(* IEC 61131-3 sources: axopen.integrations.hwc/app/SystemConstants, 2 files *)

(* ---- plc_line_HwIdentifiers.st ---- *)
CONFIGURATION HardwareIDs
    VAR_GLOBAL CONSTANT
        BNIPNT507005Z040_HwID : UINT := UINT#394;
        BNIPNT507005Z040_BIS_M_4XX_045_1_BIS_M_4XX_045_HwID : UINT := UINT#397;
        BNIPNT507005Z040_BNIPNT507005Z040_HwID : UINT := UINT#396;
        BNIPNT507005Z040_BNIPNT507005Z040_BNI_PNT_507_005_Z040_HwID : UINT := UINT#401;
        BNIPNT507005Z040_BNIPNT507005Z040_profinet_HwID : UINT := UINT#391;
        BNIPNT507005Z040_BNIPNT507005Z040_profinet_port_1___M12_HwID : UINT := UINT#392;
        BNIPNT507005Z040_BNIPNT507005Z040_profinet_port_2___M12_HwID : UINT := UINT#393;
        BNIPNT507005Z040_Rack_HwID : UINT := UINT#395;
        BNIPNT507005Z040_Standard_I_O_2_Standard_I_O_HwID : UINT := UINT#400;
        BNIPNT507005Z040_Standard_I_O_3_Standard_I_O_HwID : UINT := UINT#399;
        BNIPNT507005Z040_Standard_I_O_4_Standard_I_O_HwID : UINT := UINT#398;
        KRC4_HwID : UINT := UINT#467;
        KRC4_512_digital_in_and_outputs_1_512_digital_in__and_outputs_HwID : UINT := UINT#470;
        KRC4_KRC4_HwID : UINT := UINT#469;
        KRC4_KRC4_KRC4_ProfiNet_5_0_HwID : UINT := UINT#471;
        KRC4_KRC4_profinet_HwID : UINT := UINT#465;
        KRC4_KRC4_profinet_Port1_HwID : UINT := UINT#466;
        KRC4_Rack_HwID : UINT := UINT#468;
        OmniCore_HwID : UINT := UINT#337;
        OmniCore_DI_64_bytes_DI_64_bytes_HwID : UINT := UINT#341;
        OmniCore_DO_64_bytes_DO_64_bytes_HwID : UINT := UINT#340;
        OmniCore_OmniCore_HwID : UINT := UINT#339;
        OmniCore_OmniCore_OmniCore_Standard_PROFINET_Device_HwID : UINT := UINT#342;
        OmniCore_OmniCore_profinet_HwID : UINT := UINT#335;
        OmniCore_OmniCore_profinet_Network_Port_1_HwID : UINT := UINT#336;
        OmniCore_Rack_HwID : UINT := UINT#338;
        PROFINET_IO_System_HwID : UINT := UINT#256;
        RobotBasicIO_HwID : UINT := UINT#345;
        RobotBasicIO_DI_64_bytes_DI_64_bytes_HwID : UINT := UINT#349;
        RobotBasicIO_DO_64_bytes_DO_64_bytes_HwID : UINT := UINT#348;
        RobotBasicIO_Rack_HwID : UINT := UINT#346;
        RobotBasicIO_RobotBasicIO_HwID : UINT := UINT#347;
        RobotBasicIO_RobotBasicIO_Robot_Basic_Device_HwID : UINT := UINT#350;
        RobotBasicIO_RobotBasicIO_profinet_HwID : UINT := UINT#343;
        RobotBasicIO_RobotBasicIO_profinet_Network_Port_HwID : UINT := UINT#344;
        SFK_HwID : UINT := UINT#305;
        SFK_F_Modul_not_used_1_ID_FMod_NotUsed_HwID : UINT := UINT#311;
        SFK_Input_24_Words_ID_InMod_24Words_HwID : UINT := UINT#309;
        SFK_Output_21_Words_ID_OutMod_21Words_HwID : UINT := UINT#308;
        SFK_ParamCh_IDN_1_ID_PaCh_5Words_HwID : UINT := UINT#310;
        SFK_Rack_HwID : UINT := UINT#306;
        SFK_SFK_HwID : UINT := UINT#307;
        SFK_SFK_DAP_1_HwID : UINT := UINT#312;
        SFK_SFK_profinet_HwID : UINT := UINT#302;
        SFK_SFK_profinet_Port_1___RJ45_HwID : UINT := UINT#303;
        SFK_SFK_profinet_Port_2___RJ45_HwID : UINT := UINT#304;
        ST3_indradrive_HwID : UINT := UINT#293;
        ST3_indradrive_F_Modul_not_used_1_ID_FMod_NotUsed_HwID : UINT := UINT#299;
        ST3_indradrive_Input_9_Words_1_ID_InMod_9Words_HwID : UINT := UINT#297;
        ST3_indradrive_Output_13_Words_1_ID_OutMod_13Words_HwID : UINT := UINT#296;
        ST3_indradrive_ParamCh_IDN_1_ID_PaCh_5Words_HwID : UINT := UINT#298;
        ST3_indradrive_Rack_HwID : UINT := UINT#294;
        ST3_indradrive_ST3_indradrive_HwID : UINT := UINT#295;
        ST3_indradrive_ST3_indradrive_DAP_1_HwID : UINT := UINT#300;
        ST3_indradrive_ST3_indradrive_profinet_HwID : UINT := UINT#290;
        ST3_indradrive_ST3_indradrive_profinet_Port_1___RJ45_HwID : UINT := UINT#291;
        ST3_indradrive_ST3_indradrive_profinet_Port_2___RJ45_HwID : UINT := UINT#292;
        TZ535_PN_HwID : UINT := UINT#316;
        TZ535_PN_In_Out_64_byte_1_In_Out__64_byte_HwID : UINT := UINT#319;
        TZ535_PN_Rack_HwID : UINT := UINT#317;
        TZ535_PN_TZ535_PN_HwID : UINT := UINT#318;
        TZ535_PN_TZ535_PN_2D_TZ535_PNPROFINET_IO_HwID : UINT := UINT#320;
        TZ535_PN_TZ535_PN_profinet_HwID : UINT := UINT#313;
        TZ535_PN_TZ535_PN_profinet_Port_1_HwID : UINT := UINT#314;
        TZ535_PN_TZ535_PN_profinet_Port_2_HwID : UINT := UINT#315;
        URIODev1_HwID : UINT := UINT#276;
        URIODev1_1_HwID : UINT := UINT#259;
        URIODev1_1_10_O2T_General_Purpose_Registers_2_1_10_O2T_General_Purpose_Registers_2_HwID : UINT := UINT#262;
        URIODev1_1_1_T2O_State_1_1_T2O_State_HwID : UINT := UINT#271;
        URIODev1_1_2_T2O_IO_1_2_T2O_IO_HwID : UINT := UINT#270;
        URIODev1_1_3_T2O_Joints_1_3_T2O_Joints_HwID : UINT := UINT#269;
        URIODev1_1_4_T2O_TCP_1_4_T2O_TCP_HwID : UINT := UINT#268;
        URIODev1_1_5_T2O_General_Purpose_Bit_Registers_1_5_T2O_General_Purpose_Bit_Registers_HwID : UINT := UINT#267;
        URIODev1_1_6_T2O_General_Purpose_Int_Registers_1_6_T2O_General_Purpose_Int_Registers_HwID : UINT := UINT#266;
        URIODev1_1_7_T2O_General_Purpose_Float_Registers_1_7_T2O_General_Purpose_Float_Registers_HwID : UINT := UINT#265;
        URIODev1_1_8_O2T_Robot_IO_1_8_O2T_Robot_IO_HwID : UINT := UINT#264;
        URIODev1_1_9_O2T_General_Purpose_Registers_1_1_9_O2T_General_Purpose_Registers_1_HwID : UINT := UINT#263;
        URIODev1_1_PROFIsafe_1_Module_Access_Point_HwID : UINT := UINT#272;
        URIODev1_1_Rack_HwID : UINT := UINT#260;
        URIODev1_1_URIODev1_1_HwID : UINT := UINT#261;
        URIODev1_1_URIODev1_1_V1_0_HwID : UINT := UINT#273;
        URIODev1_1_URIODev1_1_profinet_HwID : UINT := UINT#257;
        URIODev1_1_URIODev1_1_profinet_RJ45_10_100_MBit_s_HwID : UINT := UINT#258;
        URIODev1_10_O2T_General_Purpose_Registers_2_1_10_O2T_General_Purpose_Registers_2_HwID : UINT := UINT#279;
        URIODev1_1_T2O_State_1_1_T2O_State_HwID : UINT := UINT#288;
        URIODev1_2_T2O_IO_1_2_T2O_IO_HwID : UINT := UINT#287;
        URIODev1_3_T2O_Joints_1_3_T2O_Joints_HwID : UINT := UINT#286;
        URIODev1_4_T2O_TCP_1_4_T2O_TCP_HwID : UINT := UINT#285;
        URIODev1_5_T2O_General_Purpose_Bit_Registers_1_5_T2O_General_Purpose_Bit_Registers_HwID : UINT := UINT#284;
        URIODev1_6_T2O_General_Purpose_Int_Registers_1_6_T2O_General_Purpose_Int_Registers_HwID : UINT := UINT#283;
        URIODev1_7_T2O_General_Purpose_Float_Registers_1_7_T2O_General_Purpose_Float_Registers_HwID : UINT := UINT#282;
        URIODev1_8_O2T_Robot_IO_1_8_O2T_Robot_IO_HwID : UINT := UINT#281;
        URIODev1_9_O2T_General_Purpose_Registers_1_1_9_O2T_General_Purpose_Registers_1_HwID : UINT := UINT#280;
        URIODev1_Rack_HwID : UINT := UINT#277;
        URIODev1_URIODev1_HwID : UINT := UINT#278;
        URIODev1_URIODev1_V1_0_HwID : UINT := UINT#289;
        URIODev1_URIODev1_profinet_HwID : UINT := UINT#274;
        URIODev1_URIODev1_profinet_RJ45_10_100_MBit_s_HwID : UINT := UINT#275;
        aventics_HwID : UINT := UINT#405;
        aventics_Rack_HwID : UINT := UINT#406;
        aventics_Valve_driver_2_valves_1_Valve_driver_2_valves_2_HwID : UINT := UINT#408;
        aventics_Valve_driver_3_valves_1_Valve_driver_3_valves_3_HwID : UINT := UINT#411;
        aventics_Valve_driver_4_valves_1_Valve_driver_4_valves_4_HwID : UINT := UINT#412;
        aventics_Valve_driver_4_valves_2_Valve_driver_4_valves_4_HwID : UINT := UINT#410;
        aventics_Valve_driver_4_valves_3_Valve_driver_4_valves_4_HwID : UINT := UINT#409;
        aventics_aventics_HwID : UINT := UINT#407;
        aventics_aventics_AES_Modul_HwID : UINT := UINT#413;
        aventics_aventics_profinet_HwID : UINT := UINT#402;
        aventics_aventics_profinet_Port_1_HwID : UINT := UINT#403;
        aventics_aventics_profinet_Port_2_HwID : UINT := UINT#404;
        cmmtas_HwID : UINT := UINT#456;
        cmmtas_Rack_HwID : UINT := UINT#457;
        cmmtas_SiemensTelegram111_PZD_12_12_HwID : UINT := UINT#462;
        cmmtas_SiemensTelegram750_PZD_4_1_HwID : UINT := UINT#463;
        cmmtas_cmmtas_HwID : UINT := UINT#458;
        cmmtas_cmmtas_CMMT_AS_____MP_HwID : UINT := UINT#464;
        cmmtas_cmmtas_DoServo_HwID : UINT := UINT#459;
        cmmtas_cmmtas_DoServo_Module_Access_Point_HwID : UINT := UINT#461;
        cmmtas_cmmtas_empty_submodule_HwID : UINT := UINT#460;
        cmmtas_cmmtas_profinet_HwID : UINT := UINT#453;
        cmmtas_cmmtas_profinet_Port_1_HwID : UINT := UINT#454;
        cmmtas_cmmtas_profinet_Port_2_HwID : UINT := UINT#455;
        et200sp_HwID : UINT := UINT#438;
        et200sp_1_HwID : UINT := UINT#427;
        et200sp_1_DI_ST_1_DI_8x24VDC_ST_V1_1_HwID : UINT := UINT#432;
        et200sp_1_DI_ST_2_DI_8x24VDC_ST_V1_1_HwID : UINT := UINT#431;
        et200sp_1_DQ_ST_1_DQ_8x24VDC_0_5A_ST_V1_1_HwID : UINT := UINT#433;
        et200sp_1_Rack_HwID : UINT := UINT#428;
        et200sp_1_Server_module_V1_1_Server_module_V1_1_0_bytes_HwID : UINT := UINT#430;
        et200sp_1_et200sp_1_HwID : UINT := UINT#429;
        et200sp_1_et200sp_1_IM_155_6_PN_ST_V3_3_HwID : UINT := UINT#434;
        et200sp_1_et200sp_1_Port_1_2xRJ45_HwID : UINT := UINT#425;
        et200sp_1_et200sp_1_Port_2_2xRJ45_HwID : UINT := UINT#426;
        et200sp_1_et200sp_1_profinet_HwID : UINT := UINT#424;
        et200sp_CM_4xIO_Link_V2_2_144I_128O_1_CM_4xIO_Link_V2_2_144I_128O_HwID : UINT := UINT#442;
        et200sp_Rack_HwID : UINT := UINT#439;
        et200sp_Server_module_V1_1_Server_module_V1_1_0_bytes_HwID : UINT := UINT#441;
        et200sp_et200sp_HwID : UINT := UINT#440;
        et200sp_et200sp_IM_155_6_PN_ST_V4_2_HwID : UINT := UINT#443;
        et200sp_et200sp_Port_1_2xRJ45_HwID : UINT := UINT#436;
        et200sp_et200sp_Port_2_2xRJ45_HwID : UINT := UINT#437;
        et200sp_et200sp_profinet_HwID : UINT := UINT#435;
        festocpx_HwID : UINT := UINT#417;
        festocpx_FB43_PNIO_Module_1_FB43_PNIO_Module_HwID : UINT := UINT#422;
        festocpx_MPA1S_VMPA1_FB_EMG_8_1_MPA1G_VMPA1_FB_EMG_8_8DO_HwID : UINT := UINT#420;
        festocpx_MPA1S_VMPA1_FB_EMS_8_MPA1S_VMPA1_FB_EMS_8_8DO_HwID : UINT := UINT#421;
        festocpx_Rack_HwID : UINT := UINT#418;
        festocpx_festocpx_HwID : UINT := UINT#419;
        festocpx_festocpx_CPX_Rev_50_HwID : UINT := UINT#423;
        festocpx_festocpx_profinet_HwID : UINT := UINT#414;
        festocpx_festocpx_profinet_Port_1_HwID : UINT := UINT#415;
        festocpx_festocpx_profinet_Port_2_HwID : UINT := UINT#416;
        is7600_HwID : UINT := UINT#353;
        is7600_Acquisition_Control_Acquisition_Control_HwID : UINT := UINT#363;
        is7600_Acquisition_Status_Acquisition_Status_HwID : UINT := UINT#359;
        is7600_Command_Control_Command_Control_HwID : UINT := UINT#360;
        is7600_Inspection_Control_Inspection_Control_HwID : UINT := UINT#362;
        is7600_Inspection_Status_Inspection_Status_HwID : UINT := UINT#358;
        is7600_Rack_HwID : UINT := UINT#354;
        is7600_Result_Data_64_bytes_Results___64_bytes_HwID : UINT := UINT#356;
        is7600_SoftEvent_Control_SoftEvent_Control_HwID : UINT := UINT#361;
        is7600_User_Data_64_bytes_User_Data___64_bytes_HwID : UINT := UINT#357;
        is7600_is7600_HwID : UINT := UINT#355;
        is7600_is7600_In_Sight_IS79XX_IS75XX_CC_B_HwID : UINT := UINT#364;
        is7600_is7600_profinet_HwID : UINT := UINT#351;
        is7600_is7600_profinet_Port_1_HwID : UINT := UINT#352;
        plc_line_HwID : UINT := UINT#32;
        plc_line_Rail_0_HwID : UINT := UINT#301;
        plc_line_plc_line_HwID : UINT := UINT#48;
        plc_line_plc_line__plc_line_HwID : UINT := UINT#49;
        plc_line_plc_line_CPU_display_1_HwID : UINT := UINT#54;
        plc_line_plc_line_CPU_exec_unit_1_HwID : UINT := UINT#52;
        plc_line_plc_line_Card_reader_writer_1_HwID : UINT := UINT#51;
        plc_line_plc_line_DP_interface_1_HwID : UINT := UINT#60;
        plc_line_plc_line_LicenseManager_1_HwID : UINT := UINT#42;
        plc_line_plc_line_OPC_UA_1_HwID : UINT := UINT#117;
        plc_line_plc_line_PROFINET_interface_2_HwID : UINT := UINT#72;
        plc_line_plc_line_PROFINET_interface_2_Port_1_HwID : UINT := UINT#73;
        plc_line_plc_line_Virtual_communication_interface_HwID : UINT := UINT#135;
        plc_line_plc_line_plc_line_HwID : UINT := UINT#50;
        plc_line_plc_line_profinet_HwID : UINT := UINT#64;
        plc_line_plc_line_profinet_Port1_HwID : UINT := UINT#65;
        plc_line_plc_line_profinet_Port2_HwID : UINT := UINT#66;
        reader_st1_HwID : UINT := UINT#380;
        reader_st1_Acquisition_Control_Acquisition_Control_HwID : UINT := UINT#389;
        reader_st1_Acquisition_Status_Acquisition_Status_HwID : UINT := UINT#388;
        reader_st1_Rack_HwID : UINT := UINT#381;
        reader_st1_Result_Data___64_bytes_1_Result_Data___64_bytes_HwID : UINT := UINT#383;
        reader_st1_Results_Control_Results_Control_HwID : UINT := UINT#387;
        reader_st1_Results_Status_Results_Status_HwID : UINT := UINT#386;
        reader_st1_Soft_Event_Control_Soft_Event_Control_HwID : UINT := UINT#385;
        reader_st1_User_Data___64_bytes_1_User_Data___64_bytes_HwID : UINT := UINT#384;
        reader_st1_reader_st1_HwID : UINT := UINT#382;
        reader_st1_reader_st1_DataMan_280_CC_B_HwID : UINT := UINT#390;
        reader_st1_reader_st1_profinet_HwID : UINT := UINT#378;
        reader_st1_reader_st1_profinet_Port_1_HwID : UINT := UINT#379;
        reader_st2_HwID : UINT := UINT#367;
        reader_st2_Acquisition_Control_Acquisition_Control_HwID : UINT := UINT#376;
        reader_st2_Acquisition_Status_Acquisition_Status_HwID : UINT := UINT#375;
        reader_st2_Rack_HwID : UINT := UINT#368;
        reader_st2_Result_Data_64_bytes_Result_Data___64_bytes_HwID : UINT := UINT#370;
        reader_st2_Results_Control_Results_Control_HwID : UINT := UINT#374;
        reader_st2_Results_Status_Results_Status_HwID : UINT := UINT#373;
        reader_st2_Soft_Event_Control_Soft_Event_Control_HwID : UINT := UINT#372;
        reader_st2_User_Data_64_bytes_User_Data___64_bytes_HwID : UINT := UINT#371;
        reader_st2_reader_st2_HwID : UINT := UINT#369;
        reader_st2_reader_st2_DataMan_300_HwID : UINT := UINT#377;
        reader_st2_reader_st2_profinet_HwID : UINT := UINT#365;
        reader_st2_reader_st2_profinet_Port_1_HwID : UINT := UINT#366;
        rf186c_HwID : UINT := UINT#447;
        rf186c_Rack_HwID : UINT := UINT#448;
        rf186c_Reader_1__Reader__HwID : UINT := UINT#450;
        rf186c_rf186c_HwID : UINT := UINT#449;
        rf186c_rf186c_CM_1__Communication__HwID : UINT := UINT#451;
        rf186c_rf186c_RF186C___V2_x_HwID : UINT := UINT#452;
        rf186c_rf186c_profinet_HwID : UINT := UINT#444;
        rf186c_rf186c_profinet_Port_1_HwID : UINT := UINT#445;
        rf186c_rf186c_profinet_Port_2_HwID : UINT := UINT#446;
        wp462_t1_rh_deso_HwID : UINT := UINT#323;
        wp462_t1_rh_deso_Input_1_byte_1_Input_1_byte_HwID : UINT := UINT#333;
        wp462_t1_rh_deso_Input_1_byte_2_Input_1_byte_HwID : UINT := UINT#332;
        wp462_t1_rh_deso_Input_1_word_1_Input_1_word_HwID : UINT := UINT#330;
        wp462_t1_rh_deso_Input_1_word_2_Input_1_word_HwID : UINT := UINT#328;
        wp462_t1_rh_deso_Input_2_word_1_Input_2_word_HwID : UINT := UINT#331;
        wp462_t1_rh_deso_Input_2_word_2_Input_2_word_HwID : UINT := UINT#329;
        wp462_t1_rh_deso_Output_1_byte_1_Output_1_byte_HwID : UINT := UINT#327;
        wp462_t1_rh_deso_Output_1_byte_2_Output_1_byte_HwID : UINT := UINT#326;
        wp462_t1_rh_deso_Rack_HwID : UINT := UINT#324;
        wp462_t1_rh_deso_wp462_t1_rh_deso_HwID : UINT := UINT#325;
        wp462_t1_rh_deso_wp462_t1_rh_deso_RT_HwID : UINT := UINT#334;
        wp462_t1_rh_deso_wp462_t1_rh_deso_profinet_HwID : UINT := UINT#321;
        wp462_t1_rh_deso_wp462_t1_rh_deso_profinet_Port_1_HwID : UINT := UINT#322;

    END_VAR
END_CONFIGURATION

(* ---- plc_line_IoAddresses.st ---- *)
CONFIGURATION IoAddresses
    VAR_GLOBAL
        BNIPNT507005Z040_BIS_M_4XX_045_1_InputAddress_0 AT %IW1484: WORD;
        BNIPNT507005Z040_BIS_M_4XX_045_1_InputAddress_1 AT %IW1486: WORD;
        BNIPNT507005Z040_BIS_M_4XX_045_1_InputAddress_2 AT %IW1488: WORD;
        BNIPNT507005Z040_BIS_M_4XX_045_1_InputAddress_3 AT %IW1490: WORD;
        BNIPNT507005Z040_BIS_M_4XX_045_1_InputAddress_4 AT %IW1492: WORD;
        BNIPNT507005Z040_BIS_M_4XX_045_1_OutputAddress_0 AT %QW941: WORD;
        BNIPNT507005Z040_BIS_M_4XX_045_1_OutputAddress_1 AT %QW943: WORD;
        BNIPNT507005Z040_BIS_M_4XX_045_1_OutputAddress_2 AT %QW945: WORD;
        BNIPNT507005Z040_BIS_M_4XX_045_1_OutputAddress_3 AT %QW947: WORD;
        BNIPNT507005Z040_BIS_M_4XX_045_1_OutputAddress_4 AT %QW949: WORD;
        KRC4_512_digital_in_and_outputs_1_InputAddress_0 AT %IL1407: LWORD;
        KRC4_512_digital_in_and_outputs_1_InputAddress_1 AT %IL1415: LWORD;
        KRC4_512_digital_in_and_outputs_1_InputAddress_2 AT %IL1423: LWORD;
        KRC4_512_digital_in_and_outputs_1_InputAddress_3 AT %IL1431: LWORD;
        KRC4_512_digital_in_and_outputs_1_InputAddress_4 AT %IL1439: LWORD;
        KRC4_512_digital_in_and_outputs_1_InputAddress_5 AT %IL1447: LWORD;
        KRC4_512_digital_in_and_outputs_1_InputAddress_6 AT %IL1455: LWORD;
        KRC4_512_digital_in_and_outputs_1_InputAddress_7 AT %IL1463: LWORD;
        KRC4_512_digital_in_and_outputs_1_OutputAddress_0 AT %QL870: LWORD;
        KRC4_512_digital_in_and_outputs_1_OutputAddress_1 AT %QL878: LWORD;
        KRC4_512_digital_in_and_outputs_1_OutputAddress_2 AT %QL886: LWORD;
        KRC4_512_digital_in_and_outputs_1_OutputAddress_3 AT %QL894: LWORD;
        KRC4_512_digital_in_and_outputs_1_OutputAddress_4 AT %QL902: LWORD;
        KRC4_512_digital_in_and_outputs_1_OutputAddress_5 AT %QL910: LWORD;
        KRC4_512_digital_in_and_outputs_1_OutputAddress_6 AT %QL918: LWORD;
        KRC4_512_digital_in_and_outputs_1_OutputAddress_7 AT %QL926: LWORD;
        OmniCore_DI_64_bytes_InputAddress_0 AT %IL1124: LWORD;
        OmniCore_DI_64_bytes_InputAddress_1 AT %IL1132: LWORD;
        OmniCore_DI_64_bytes_InputAddress_2 AT %IL1140: LWORD;
        OmniCore_DI_64_bytes_InputAddress_3 AT %IL1148: LWORD;
        OmniCore_DI_64_bytes_InputAddress_4 AT %IL1156: LWORD;
        OmniCore_DI_64_bytes_InputAddress_5 AT %IL1164: LWORD;
        OmniCore_DI_64_bytes_InputAddress_6 AT %IL1172: LWORD;
        OmniCore_DI_64_bytes_InputAddress_7 AT %IL1180: LWORD;
        OmniCore_DO_64_bytes_OutputAddress_0 AT %QL602: LWORD;
        OmniCore_DO_64_bytes_OutputAddress_1 AT %QL610: LWORD;
        OmniCore_DO_64_bytes_OutputAddress_2 AT %QL618: LWORD;
        OmniCore_DO_64_bytes_OutputAddress_3 AT %QL626: LWORD;
        OmniCore_DO_64_bytes_OutputAddress_4 AT %QL634: LWORD;
        OmniCore_DO_64_bytes_OutputAddress_5 AT %QL642: LWORD;
        OmniCore_DO_64_bytes_OutputAddress_6 AT %QL650: LWORD;
        OmniCore_DO_64_bytes_OutputAddress_7 AT %QL658: LWORD;
        RobotBasicIO_DI_64_bytes_InputAddress_0 AT %IL1188: LWORD;
        RobotBasicIO_DI_64_bytes_InputAddress_1 AT %IL1196: LWORD;
        RobotBasicIO_DI_64_bytes_InputAddress_2 AT %IL1204: LWORD;
        RobotBasicIO_DI_64_bytes_InputAddress_3 AT %IL1212: LWORD;
        RobotBasicIO_DI_64_bytes_InputAddress_4 AT %IL1220: LWORD;
        RobotBasicIO_DI_64_bytes_InputAddress_5 AT %IL1228: LWORD;
        RobotBasicIO_DI_64_bytes_InputAddress_6 AT %IL1236: LWORD;
        RobotBasicIO_DI_64_bytes_InputAddress_7 AT %IL1244: LWORD;
        RobotBasicIO_DO_64_bytes_OutputAddress_0 AT %QL666: LWORD;
        RobotBasicIO_DO_64_bytes_OutputAddress_1 AT %QL674: LWORD;
        RobotBasicIO_DO_64_bytes_OutputAddress_2 AT %QL682: LWORD;
        RobotBasicIO_DO_64_bytes_OutputAddress_3 AT %QL690: LWORD;
        RobotBasicIO_DO_64_bytes_OutputAddress_4 AT %QL698: LWORD;
        RobotBasicIO_DO_64_bytes_OutputAddress_5 AT %QL706: LWORD;
        RobotBasicIO_DO_64_bytes_OutputAddress_6 AT %QL714: LWORD;
        RobotBasicIO_DO_64_bytes_OutputAddress_7 AT %QL722: LWORD;
        SFK_Input_24_Words_InputAddress_0 AT %IL988: LWORD;
        SFK_Input_24_Words_InputAddress_1 AT %IL996: LWORD;
        SFK_Input_24_Words_InputAddress_2 AT %IL1004: LWORD;
        SFK_Input_24_Words_InputAddress_3 AT %IL1012: LWORD;
        SFK_Input_24_Words_InputAddress_4 AT %IL1020: LWORD;
        SFK_Input_24_Words_InputAddress_5 AT %IL1028: LWORD;
        SFK_Output_21_Words_OutputAddress_0 AT %QW484: WORD;
        SFK_Output_21_Words_OutputAddress_1 AT %QW486: WORD;
        SFK_Output_21_Words_OutputAddress_2 AT %QW488: WORD;
        SFK_Output_21_Words_OutputAddress_3 AT %QW490: WORD;
        SFK_Output_21_Words_OutputAddress_4 AT %QW492: WORD;
        SFK_Output_21_Words_OutputAddress_5 AT %QW494: WORD;
        SFK_Output_21_Words_OutputAddress_6 AT %QW496: WORD;
        SFK_Output_21_Words_OutputAddress_7 AT %QW498: WORD;
        SFK_Output_21_Words_OutputAddress_8 AT %QW500: WORD;
        SFK_Output_21_Words_OutputAddress_9 AT %QW502: WORD;
        SFK_Output_21_Words_OutputAddress_10 AT %QW504: WORD;
        SFK_Output_21_Words_OutputAddress_11 AT %QW506: WORD;
        SFK_Output_21_Words_OutputAddress_12 AT %QW508: WORD;
        SFK_Output_21_Words_OutputAddress_13 AT %QW510: WORD;
        SFK_Output_21_Words_OutputAddress_14 AT %QW512: WORD;
        SFK_Output_21_Words_OutputAddress_15 AT %QW514: WORD;
        SFK_Output_21_Words_OutputAddress_16 AT %QW516: WORD;
        SFK_Output_21_Words_OutputAddress_17 AT %QW518: WORD;
        SFK_Output_21_Words_OutputAddress_18 AT %QW520: WORD;
        SFK_Output_21_Words_OutputAddress_19 AT %QW522: WORD;
        SFK_Output_21_Words_OutputAddress_20 AT %QW524: WORD;
        SFK_ParamCh_IDN_1_InputAddress_0 AT %IW1036: WORD;
        SFK_ParamCh_IDN_1_InputAddress_1 AT %IW1038: WORD;
        SFK_ParamCh_IDN_1_InputAddress_2 AT %IW1040: WORD;
        SFK_ParamCh_IDN_1_InputAddress_3 AT %IW1042: WORD;
        SFK_ParamCh_IDN_1_InputAddress_4 AT %IW1044: WORD;
        SFK_ParamCh_IDN_1_OutputAddress_0 AT %QW526: WORD;
        SFK_ParamCh_IDN_1_OutputAddress_1 AT %QW528: WORD;
        SFK_ParamCh_IDN_1_OutputAddress_2 AT %QW530: WORD;
        SFK_ParamCh_IDN_1_OutputAddress_3 AT %QW532: WORD;
        SFK_ParamCh_IDN_1_OutputAddress_4 AT %QW534: WORD;
        ST3_indradrive_Input_9_Words_1_InputAddress_0 AT %IW960: WORD;
        ST3_indradrive_Input_9_Words_1_InputAddress_1 AT %IW962: WORD;
        ST3_indradrive_Input_9_Words_1_InputAddress_2 AT %IW964: WORD;
        ST3_indradrive_Input_9_Words_1_InputAddress_3 AT %IW966: WORD;
        ST3_indradrive_Input_9_Words_1_InputAddress_4 AT %IW968: WORD;
        ST3_indradrive_Input_9_Words_1_InputAddress_5 AT %IW970: WORD;
        ST3_indradrive_Input_9_Words_1_InputAddress_6 AT %IW972: WORD;
        ST3_indradrive_Input_9_Words_1_InputAddress_7 AT %IW974: WORD;
        ST3_indradrive_Input_9_Words_1_InputAddress_8 AT %IW976: WORD;
        ST3_indradrive_Output_13_Words_1_OutputAddress_0 AT %QW448: WORD;
        ST3_indradrive_Output_13_Words_1_OutputAddress_1 AT %QW450: WORD;
        ST3_indradrive_Output_13_Words_1_OutputAddress_2 AT %QW452: WORD;
        ST3_indradrive_Output_13_Words_1_OutputAddress_3 AT %QW454: WORD;
        ST3_indradrive_Output_13_Words_1_OutputAddress_4 AT %QW456: WORD;
        ST3_indradrive_Output_13_Words_1_OutputAddress_5 AT %QW458: WORD;
        ST3_indradrive_Output_13_Words_1_OutputAddress_6 AT %QW460: WORD;
        ST3_indradrive_Output_13_Words_1_OutputAddress_7 AT %QW462: WORD;
        ST3_indradrive_Output_13_Words_1_OutputAddress_8 AT %QW464: WORD;
        ST3_indradrive_Output_13_Words_1_OutputAddress_9 AT %QW466: WORD;
        ST3_indradrive_Output_13_Words_1_OutputAddress_10 AT %QW468: WORD;
        ST3_indradrive_Output_13_Words_1_OutputAddress_11 AT %QW470: WORD;
        ST3_indradrive_Output_13_Words_1_OutputAddress_12 AT %QW472: WORD;
        ST3_indradrive_ParamCh_IDN_1_InputAddress_0 AT %IW978: WORD;
        ST3_indradrive_ParamCh_IDN_1_InputAddress_1 AT %IW980: WORD;
        ST3_indradrive_ParamCh_IDN_1_InputAddress_2 AT %IW982: WORD;
        ST3_indradrive_ParamCh_IDN_1_InputAddress_3 AT %IW984: WORD;
        ST3_indradrive_ParamCh_IDN_1_InputAddress_4 AT %IW986: WORD;
        ST3_indradrive_ParamCh_IDN_1_OutputAddress_0 AT %QW474: WORD;
        ST3_indradrive_ParamCh_IDN_1_OutputAddress_1 AT %QW476: WORD;
        ST3_indradrive_ParamCh_IDN_1_OutputAddress_2 AT %QW478: WORD;
        ST3_indradrive_ParamCh_IDN_1_OutputAddress_3 AT %QW480: WORD;
        ST3_indradrive_ParamCh_IDN_1_OutputAddress_4 AT %QW482: WORD;
        TZ535_PN_In_Out_64_byte_1_InputAddress_0 AT %IL1046: LWORD;
        TZ535_PN_In_Out_64_byte_1_InputAddress_1 AT %IL1054: LWORD;
        TZ535_PN_In_Out_64_byte_1_InputAddress_2 AT %IL1062: LWORD;
        TZ535_PN_In_Out_64_byte_1_InputAddress_3 AT %IL1070: LWORD;
        TZ535_PN_In_Out_64_byte_1_InputAddress_4 AT %IL1078: LWORD;
        TZ535_PN_In_Out_64_byte_1_InputAddress_5 AT %IL1086: LWORD;
        TZ535_PN_In_Out_64_byte_1_InputAddress_6 AT %IL1094: LWORD;
        TZ535_PN_In_Out_64_byte_1_InputAddress_7 AT %IL1102: LWORD;
        TZ535_PN_In_Out_64_byte_1_OutputAddress_0 AT %QL536: LWORD;
        TZ535_PN_In_Out_64_byte_1_OutputAddress_1 AT %QL544: LWORD;
        TZ535_PN_In_Out_64_byte_1_OutputAddress_2 AT %QL552: LWORD;
        TZ535_PN_In_Out_64_byte_1_OutputAddress_3 AT %QL560: LWORD;
        TZ535_PN_In_Out_64_byte_1_OutputAddress_4 AT %QL568: LWORD;
        TZ535_PN_In_Out_64_byte_1_OutputAddress_5 AT %QL576: LWORD;
        TZ535_PN_In_Out_64_byte_1_OutputAddress_6 AT %QL584: LWORD;
        TZ535_PN_In_Out_64_byte_1_OutputAddress_7 AT %QL592: LWORD;
        URIODev1_10_O2T_General_Purpose_Registers_2_1_OutputAddress_0 AT %QD224: DWORD;
        URIODev1_10_O2T_General_Purpose_Registers_2_1_OutputAddress_1 AT %QD228: DWORD;
        URIODev1_10_O2T_General_Purpose_Registers_2_1_OutputAddress_2 AT %QD232: DWORD;
        URIODev1_10_O2T_General_Purpose_Registers_2_1_OutputAddress_3 AT %QD236: DWORD;
        URIODev1_10_O2T_General_Purpose_Registers_2_1_OutputAddress_4 AT %QD240: DWORD;
        URIODev1_10_O2T_General_Purpose_Registers_2_1_OutputAddress_5 AT %QD244: DWORD;
        URIODev1_10_O2T_General_Purpose_Registers_2_1_OutputAddress_6 AT %QD248: DWORD;
        URIODev1_10_O2T_General_Purpose_Registers_2_1_OutputAddress_7 AT %QD252: DWORD;
        URIODev1_10_O2T_General_Purpose_Registers_2_1_OutputAddress_8 AT %QD256: DWORD;
        URIODev1_10_O2T_General_Purpose_Registers_2_1_OutputAddress_9 AT %QD260: DWORD;
        URIODev1_10_O2T_General_Purpose_Registers_2_1_OutputAddress_10 AT %QD264: DWORD;
        URIODev1_10_O2T_General_Purpose_Registers_2_1_OutputAddress_11 AT %QD268: DWORD;
        URIODev1_10_O2T_General_Purpose_Registers_2_1_OutputAddress_12 AT %QD272: DWORD;
        URIODev1_10_O2T_General_Purpose_Registers_2_1_OutputAddress_13 AT %QD276: DWORD;
        URIODev1_10_O2T_General_Purpose_Registers_2_1_OutputAddress_14 AT %QD280: DWORD;
        URIODev1_10_O2T_General_Purpose_Registers_2_1_OutputAddress_15 AT %QD284: DWORD;
        URIODev1_10_O2T_General_Purpose_Registers_2_1_OutputAddress_16 AT %QD288: DWORD;
        URIODev1_10_O2T_General_Purpose_Registers_2_1_OutputAddress_17 AT %QD292: DWORD;
        URIODev1_10_O2T_General_Purpose_Registers_2_1_OutputAddress_18 AT %QD296: DWORD;
        URIODev1_10_O2T_General_Purpose_Registers_2_1_OutputAddress_19 AT %QD300: DWORD;
        URIODev1_10_O2T_General_Purpose_Registers_2_1_OutputAddress_20 AT %QD304: DWORD;
        URIODev1_10_O2T_General_Purpose_Registers_2_1_OutputAddress_21 AT %QD308: DWORD;
        URIODev1_10_O2T_General_Purpose_Registers_2_1_OutputAddress_22 AT %QD312: DWORD;
        URIODev1_10_O2T_General_Purpose_Registers_2_1_OutputAddress_23 AT %QD316: DWORD;
        URIODev1_10_O2T_General_Purpose_Registers_2_1_OutputAddress_24 AT %QD320: DWORD;
        URIODev1_1_T2O_State_1_InputAddress_0 AT %IL928: LWORD;
        URIODev1_1_T2O_State_1_InputAddress_1 AT %IL936: LWORD;
        URIODev1_1_T2O_State_1_InputAddress_2 AT %IL944: LWORD;
        URIODev1_1_T2O_State_1_InputAddress_3 AT %IL952: LWORD;
        URIODev1_2_T2O_IO_1_InputAddress_0 AT %ID860: DWORD;
        URIODev1_2_T2O_IO_1_InputAddress_1 AT %ID864: DWORD;
        URIODev1_2_T2O_IO_1_InputAddress_2 AT %ID868: DWORD;
        URIODev1_2_T2O_IO_1_InputAddress_3 AT %ID872: DWORD;
        URIODev1_2_T2O_IO_1_InputAddress_4 AT %ID876: DWORD;
        URIODev1_2_T2O_IO_1_InputAddress_5 AT %ID880: DWORD;
        URIODev1_2_T2O_IO_1_InputAddress_6 AT %ID884: DWORD;
        URIODev1_2_T2O_IO_1_InputAddress_7 AT %ID888: DWORD;
        URIODev1_2_T2O_IO_1_InputAddress_8 AT %ID892: DWORD;
        URIODev1_2_T2O_IO_1_InputAddress_9 AT %ID896: DWORD;
        URIODev1_2_T2O_IO_1_InputAddress_10 AT %ID900: DWORD;
        URIODev1_2_T2O_IO_1_InputAddress_11 AT %ID904: DWORD;
        URIODev1_2_T2O_IO_1_InputAddress_12 AT %ID908: DWORD;
        URIODev1_2_T2O_IO_1_InputAddress_13 AT %ID912: DWORD;
        URIODev1_2_T2O_IO_1_InputAddress_14 AT %ID916: DWORD;
        URIODev1_2_T2O_IO_1_InputAddress_15 AT %ID920: DWORD;
        URIODev1_2_T2O_IO_1_InputAddress_16 AT %ID924: DWORD;
        URIODev1_3_T2O_Joints_1_InputAddress_0 AT %IL756: LWORD;
        URIODev1_3_T2O_Joints_1_InputAddress_1 AT %IL764: LWORD;
        URIODev1_3_T2O_Joints_1_InputAddress_2 AT %IL772: LWORD;
        URIODev1_3_T2O_Joints_1_InputAddress_3 AT %IL780: LWORD;
        URIODev1_3_T2O_Joints_1_InputAddress_4 AT %IL788: LWORD;
        URIODev1_3_T2O_Joints_1_InputAddress_5 AT %IL796: LWORD;
        URIODev1_3_T2O_Joints_1_InputAddress_6 AT %IL804: LWORD;
        URIODev1_3_T2O_Joints_1_InputAddress_7 AT %IL812: LWORD;
        URIODev1_3_T2O_Joints_1_InputAddress_8 AT %IL820: LWORD;
        URIODev1_3_T2O_Joints_1_InputAddress_9 AT %IL828: LWORD;
        URIODev1_3_T2O_Joints_1_InputAddress_10 AT %IL836: LWORD;
        URIODev1_3_T2O_Joints_1_InputAddress_11 AT %IL844: LWORD;
        URIODev1_3_T2O_Joints_1_InputAddress_12 AT %IL852: LWORD;
        URIODev1_4_T2O_TCP_1_InputAddress_0 AT %ID680: DWORD;
        URIODev1_4_T2O_TCP_1_InputAddress_1 AT %ID684: DWORD;
        URIODev1_4_T2O_TCP_1_InputAddress_2 AT %ID688: DWORD;
        URIODev1_4_T2O_TCP_1_InputAddress_3 AT %ID692: DWORD;
        URIODev1_4_T2O_TCP_1_InputAddress_4 AT %ID696: DWORD;
        URIODev1_4_T2O_TCP_1_InputAddress_5 AT %ID700: DWORD;
        URIODev1_4_T2O_TCP_1_InputAddress_6 AT %ID704: DWORD;
        URIODev1_4_T2O_TCP_1_InputAddress_7 AT %ID708: DWORD;
        URIODev1_4_T2O_TCP_1_InputAddress_8 AT %ID712: DWORD;
        URIODev1_4_T2O_TCP_1_InputAddress_9 AT %ID716: DWORD;
        URIODev1_4_T2O_TCP_1_InputAddress_10 AT %ID720: DWORD;
        URIODev1_4_T2O_TCP_1_InputAddress_11 AT %ID724: DWORD;
        URIODev1_4_T2O_TCP_1_InputAddress_12 AT %ID728: DWORD;
        URIODev1_4_T2O_TCP_1_InputAddress_13 AT %ID732: DWORD;
        URIODev1_4_T2O_TCP_1_InputAddress_14 AT %ID736: DWORD;
        URIODev1_4_T2O_TCP_1_InputAddress_15 AT %ID740: DWORD;
        URIODev1_4_T2O_TCP_1_InputAddress_16 AT %ID744: DWORD;
        URIODev1_4_T2O_TCP_1_InputAddress_17 AT %ID748: DWORD;
        URIODev1_4_T2O_TCP_1_InputAddress_18 AT %ID752: DWORD;
        URIODev1_5_T2O_General_Purpose_Bit_Registers_1_InputAddress AT %IL672: LWORD;
        URIODev1_6_T2O_General_Purpose_Int_Registers_1_InputAddress_0 AT %IL576: LWORD;
        URIODev1_6_T2O_General_Purpose_Int_Registers_1_InputAddress_1 AT %IL584: LWORD;
        URIODev1_6_T2O_General_Purpose_Int_Registers_1_InputAddress_2 AT %IL592: LWORD;
        URIODev1_6_T2O_General_Purpose_Int_Registers_1_InputAddress_3 AT %IL600: LWORD;
        URIODev1_6_T2O_General_Purpose_Int_Registers_1_InputAddress_4 AT %IL608: LWORD;
        URIODev1_6_T2O_General_Purpose_Int_Registers_1_InputAddress_5 AT %IL616: LWORD;
        URIODev1_6_T2O_General_Purpose_Int_Registers_1_InputAddress_6 AT %IL624: LWORD;
        URIODev1_6_T2O_General_Purpose_Int_Registers_1_InputAddress_7 AT %IL632: LWORD;
        URIODev1_6_T2O_General_Purpose_Int_Registers_1_InputAddress_8 AT %IL640: LWORD;
        URIODev1_6_T2O_General_Purpose_Int_Registers_1_InputAddress_9 AT %IL648: LWORD;
        URIODev1_6_T2O_General_Purpose_Int_Registers_1_InputAddress_10 AT %IL656: LWORD;
        URIODev1_6_T2O_General_Purpose_Int_Registers_1_InputAddress_11 AT %IL664: LWORD;
        URIODev1_7_T2O_General_Purpose_Float_Registers_1_InputAddress_0 AT %IL480: LWORD;
        URIODev1_7_T2O_General_Purpose_Float_Registers_1_InputAddress_1 AT %IL488: LWORD;
        URIODev1_7_T2O_General_Purpose_Float_Registers_1_InputAddress_2 AT %IL496: LWORD;
        URIODev1_7_T2O_General_Purpose_Float_Registers_1_InputAddress_3 AT %IL504: LWORD;
        URIODev1_7_T2O_General_Purpose_Float_Registers_1_InputAddress_4 AT %IL512: LWORD;
        URIODev1_7_T2O_General_Purpose_Float_Registers_1_InputAddress_5 AT %IL520: LWORD;
        URIODev1_7_T2O_General_Purpose_Float_Registers_1_InputAddress_6 AT %IL528: LWORD;
        URIODev1_7_T2O_General_Purpose_Float_Registers_1_InputAddress_7 AT %IL536: LWORD;
        URIODev1_7_T2O_General_Purpose_Float_Registers_1_InputAddress_8 AT %IL544: LWORD;
        URIODev1_7_T2O_General_Purpose_Float_Registers_1_InputAddress_9 AT %IL552: LWORD;
        URIODev1_7_T2O_General_Purpose_Float_Registers_1_InputAddress_10 AT %IL560: LWORD;
        URIODev1_7_T2O_General_Purpose_Float_Registers_1_InputAddress_11 AT %IL568: LWORD;
        URIODev1_8_O2T_Robot_IO_1_OutputAddress_0 AT %QL424: LWORD;
        URIODev1_8_O2T_Robot_IO_1_OutputAddress_1 AT %QL432: LWORD;
        URIODev1_8_O2T_Robot_IO_1_OutputAddress_2 AT %QL440: LWORD;
        URIODev1_9_O2T_General_Purpose_Registers_1_1_OutputAddress_0 AT %QD324: DWORD;
        URIODev1_9_O2T_General_Purpose_Registers_1_1_OutputAddress_1 AT %QD328: DWORD;
        URIODev1_9_O2T_General_Purpose_Registers_1_1_OutputAddress_2 AT %QD332: DWORD;
        URIODev1_9_O2T_General_Purpose_Registers_1_1_OutputAddress_3 AT %QD336: DWORD;
        URIODev1_9_O2T_General_Purpose_Registers_1_1_OutputAddress_4 AT %QD340: DWORD;
        URIODev1_9_O2T_General_Purpose_Registers_1_1_OutputAddress_5 AT %QD344: DWORD;
        URIODev1_9_O2T_General_Purpose_Registers_1_1_OutputAddress_6 AT %QD348: DWORD;
        URIODev1_9_O2T_General_Purpose_Registers_1_1_OutputAddress_7 AT %QD352: DWORD;
        URIODev1_9_O2T_General_Purpose_Registers_1_1_OutputAddress_8 AT %QD356: DWORD;
        URIODev1_9_O2T_General_Purpose_Registers_1_1_OutputAddress_9 AT %QD360: DWORD;
        URIODev1_9_O2T_General_Purpose_Registers_1_1_OutputAddress_10 AT %QD364: DWORD;
        URIODev1_9_O2T_General_Purpose_Registers_1_1_OutputAddress_11 AT %QD368: DWORD;
        URIODev1_9_O2T_General_Purpose_Registers_1_1_OutputAddress_12 AT %QD372: DWORD;
        URIODev1_9_O2T_General_Purpose_Registers_1_1_OutputAddress_13 AT %QD376: DWORD;
        URIODev1_9_O2T_General_Purpose_Registers_1_1_OutputAddress_14 AT %QD380: DWORD;
        URIODev1_9_O2T_General_Purpose_Registers_1_1_OutputAddress_15 AT %QD384: DWORD;
        URIODev1_9_O2T_General_Purpose_Registers_1_1_OutputAddress_16 AT %QD388: DWORD;
        URIODev1_9_O2T_General_Purpose_Registers_1_1_OutputAddress_17 AT %QD392: DWORD;
        URIODev1_9_O2T_General_Purpose_Registers_1_1_OutputAddress_18 AT %QD396: DWORD;
        URIODev1_9_O2T_General_Purpose_Registers_1_1_OutputAddress_19 AT %QD400: DWORD;
        URIODev1_9_O2T_General_Purpose_Registers_1_1_OutputAddress_20 AT %QD404: DWORD;
        URIODev1_9_O2T_General_Purpose_Registers_1_1_OutputAddress_21 AT %QD408: DWORD;
        URIODev1_9_O2T_General_Purpose_Registers_1_1_OutputAddress_22 AT %QD412: DWORD;
        URIODev1_9_O2T_General_Purpose_Registers_1_1_OutputAddress_23 AT %QD416: DWORD;
        URIODev1_9_O2T_General_Purpose_Registers_1_1_OutputAddress_24 AT %QD420: DWORD;
        URIODev1_1_10_O2T_General_Purpose_Registers_2_1_OutputAddress_0 AT %QD0: DWORD;
        URIODev1_1_10_O2T_General_Purpose_Registers_2_1_OutputAddress_1 AT %QD4: DWORD;
        URIODev1_1_10_O2T_General_Purpose_Registers_2_1_OutputAddress_2 AT %QD8: DWORD;
        URIODev1_1_10_O2T_General_Purpose_Registers_2_1_OutputAddress_3 AT %QD12: DWORD;
        URIODev1_1_10_O2T_General_Purpose_Registers_2_1_OutputAddress_4 AT %QD16: DWORD;
        URIODev1_1_10_O2T_General_Purpose_Registers_2_1_OutputAddress_5 AT %QD20: DWORD;
        URIODev1_1_10_O2T_General_Purpose_Registers_2_1_OutputAddress_6 AT %QD24: DWORD;
        URIODev1_1_10_O2T_General_Purpose_Registers_2_1_OutputAddress_7 AT %QD28: DWORD;
        URIODev1_1_10_O2T_General_Purpose_Registers_2_1_OutputAddress_8 AT %QD32: DWORD;
        URIODev1_1_10_O2T_General_Purpose_Registers_2_1_OutputAddress_9 AT %QD36: DWORD;
        URIODev1_1_10_O2T_General_Purpose_Registers_2_1_OutputAddress_10 AT %QD40: DWORD;
        URIODev1_1_10_O2T_General_Purpose_Registers_2_1_OutputAddress_11 AT %QD44: DWORD;
        URIODev1_1_10_O2T_General_Purpose_Registers_2_1_OutputAddress_12 AT %QD48: DWORD;
        URIODev1_1_10_O2T_General_Purpose_Registers_2_1_OutputAddress_13 AT %QD52: DWORD;
        URIODev1_1_10_O2T_General_Purpose_Registers_2_1_OutputAddress_14 AT %QD56: DWORD;
        URIODev1_1_10_O2T_General_Purpose_Registers_2_1_OutputAddress_15 AT %QD60: DWORD;
        URIODev1_1_10_O2T_General_Purpose_Registers_2_1_OutputAddress_16 AT %QD64: DWORD;
        URIODev1_1_10_O2T_General_Purpose_Registers_2_1_OutputAddress_17 AT %QD68: DWORD;
        URIODev1_1_10_O2T_General_Purpose_Registers_2_1_OutputAddress_18 AT %QD72: DWORD;
        URIODev1_1_10_O2T_General_Purpose_Registers_2_1_OutputAddress_19 AT %QD76: DWORD;
        URIODev1_1_10_O2T_General_Purpose_Registers_2_1_OutputAddress_20 AT %QD80: DWORD;
        URIODev1_1_10_O2T_General_Purpose_Registers_2_1_OutputAddress_21 AT %QD84: DWORD;
        URIODev1_1_10_O2T_General_Purpose_Registers_2_1_OutputAddress_22 AT %QD88: DWORD;
        URIODev1_1_10_O2T_General_Purpose_Registers_2_1_OutputAddress_23 AT %QD92: DWORD;
        URIODev1_1_10_O2T_General_Purpose_Registers_2_1_OutputAddress_24 AT %QD96: DWORD;
        URIODev1_1_1_T2O_State_1_InputAddress_0 AT %IL448: LWORD;
        URIODev1_1_1_T2O_State_1_InputAddress_1 AT %IL456: LWORD;
        URIODev1_1_1_T2O_State_1_InputAddress_2 AT %IL464: LWORD;
        URIODev1_1_1_T2O_State_1_InputAddress_3 AT %IL472: LWORD;
        URIODev1_1_2_T2O_IO_1_InputAddress_0 AT %ID380: DWORD;
        URIODev1_1_2_T2O_IO_1_InputAddress_1 AT %ID384: DWORD;
        URIODev1_1_2_T2O_IO_1_InputAddress_2 AT %ID388: DWORD;
        URIODev1_1_2_T2O_IO_1_InputAddress_3 AT %ID392: DWORD;
        URIODev1_1_2_T2O_IO_1_InputAddress_4 AT %ID396: DWORD;
        URIODev1_1_2_T2O_IO_1_InputAddress_5 AT %ID400: DWORD;
        URIODev1_1_2_T2O_IO_1_InputAddress_6 AT %ID404: DWORD;
        URIODev1_1_2_T2O_IO_1_InputAddress_7 AT %ID408: DWORD;
        URIODev1_1_2_T2O_IO_1_InputAddress_8 AT %ID412: DWORD;
        URIODev1_1_2_T2O_IO_1_InputAddress_9 AT %ID416: DWORD;
        URIODev1_1_2_T2O_IO_1_InputAddress_10 AT %ID420: DWORD;
        URIODev1_1_2_T2O_IO_1_InputAddress_11 AT %ID424: DWORD;
        URIODev1_1_2_T2O_IO_1_InputAddress_12 AT %ID428: DWORD;
        URIODev1_1_2_T2O_IO_1_InputAddress_13 AT %ID432: DWORD;
        URIODev1_1_2_T2O_IO_1_InputAddress_14 AT %ID436: DWORD;
        URIODev1_1_2_T2O_IO_1_InputAddress_15 AT %ID440: DWORD;
        URIODev1_1_2_T2O_IO_1_InputAddress_16 AT %ID444: DWORD;
        URIODev1_1_3_T2O_Joints_1_InputAddress_0 AT %IL276: LWORD;
        URIODev1_1_3_T2O_Joints_1_InputAddress_1 AT %IL284: LWORD;
        URIODev1_1_3_T2O_Joints_1_InputAddress_2 AT %IL292: LWORD;
        URIODev1_1_3_T2O_Joints_1_InputAddress_3 AT %IL300: LWORD;
        URIODev1_1_3_T2O_Joints_1_InputAddress_4 AT %IL308: LWORD;
        URIODev1_1_3_T2O_Joints_1_InputAddress_5 AT %IL316: LWORD;
        URIODev1_1_3_T2O_Joints_1_InputAddress_6 AT %IL324: LWORD;
        URIODev1_1_3_T2O_Joints_1_InputAddress_7 AT %IL332: LWORD;
        URIODev1_1_3_T2O_Joints_1_InputAddress_8 AT %IL340: LWORD;
        URIODev1_1_3_T2O_Joints_1_InputAddress_9 AT %IL348: LWORD;
        URIODev1_1_3_T2O_Joints_1_InputAddress_10 AT %IL356: LWORD;
        URIODev1_1_3_T2O_Joints_1_InputAddress_11 AT %IL364: LWORD;
        URIODev1_1_3_T2O_Joints_1_InputAddress_12 AT %IL372: LWORD;
        URIODev1_1_4_T2O_TCP_1_InputAddress_0 AT %ID200: DWORD;
        URIODev1_1_4_T2O_TCP_1_InputAddress_1 AT %ID204: DWORD;
        URIODev1_1_4_T2O_TCP_1_InputAddress_2 AT %ID208: DWORD;
        URIODev1_1_4_T2O_TCP_1_InputAddress_3 AT %ID212: DWORD;
        URIODev1_1_4_T2O_TCP_1_InputAddress_4 AT %ID216: DWORD;
        URIODev1_1_4_T2O_TCP_1_InputAddress_5 AT %ID220: DWORD;
        URIODev1_1_4_T2O_TCP_1_InputAddress_6 AT %ID224: DWORD;
        URIODev1_1_4_T2O_TCP_1_InputAddress_7 AT %ID228: DWORD;
        URIODev1_1_4_T2O_TCP_1_InputAddress_8 AT %ID232: DWORD;
        URIODev1_1_4_T2O_TCP_1_InputAddress_9 AT %ID236: DWORD;
        URIODev1_1_4_T2O_TCP_1_InputAddress_10 AT %ID240: DWORD;
        URIODev1_1_4_T2O_TCP_1_InputAddress_11 AT %ID244: DWORD;
        URIODev1_1_4_T2O_TCP_1_InputAddress_12 AT %ID248: DWORD;
        URIODev1_1_4_T2O_TCP_1_InputAddress_13 AT %ID252: DWORD;
        URIODev1_1_4_T2O_TCP_1_InputAddress_14 AT %ID256: DWORD;
        URIODev1_1_4_T2O_TCP_1_InputAddress_15 AT %ID260: DWORD;
        URIODev1_1_4_T2O_TCP_1_InputAddress_16 AT %ID264: DWORD;
        URIODev1_1_4_T2O_TCP_1_InputAddress_17 AT %ID268: DWORD;
        URIODev1_1_4_T2O_TCP_1_InputAddress_18 AT %ID272: DWORD;
        URIODev1_1_5_T2O_General_Purpose_Bit_Registers_1_InputAddress AT %IL192: LWORD;
        URIODev1_1_6_T2O_General_Purpose_Int_Registers_1_InputAddress_0 AT %IL96: LWORD;
        URIODev1_1_6_T2O_General_Purpose_Int_Registers_1_InputAddress_1 AT %IL104: LWORD;
        URIODev1_1_6_T2O_General_Purpose_Int_Registers_1_InputAddress_2 AT %IL112: LWORD;
        URIODev1_1_6_T2O_General_Purpose_Int_Registers_1_InputAddress_3 AT %IL120: LWORD;
        URIODev1_1_6_T2O_General_Purpose_Int_Registers_1_InputAddress_4 AT %IL128: LWORD;
        URIODev1_1_6_T2O_General_Purpose_Int_Registers_1_InputAddress_5 AT %IL136: LWORD;
        URIODev1_1_6_T2O_General_Purpose_Int_Registers_1_InputAddress_6 AT %IL144: LWORD;
        URIODev1_1_6_T2O_General_Purpose_Int_Registers_1_InputAddress_7 AT %IL152: LWORD;
        URIODev1_1_6_T2O_General_Purpose_Int_Registers_1_InputAddress_8 AT %IL160: LWORD;
        URIODev1_1_6_T2O_General_Purpose_Int_Registers_1_InputAddress_9 AT %IL168: LWORD;
        URIODev1_1_6_T2O_General_Purpose_Int_Registers_1_InputAddress_10 AT %IL176: LWORD;
        URIODev1_1_6_T2O_General_Purpose_Int_Registers_1_InputAddress_11 AT %IL184: LWORD;
        URIODev1_1_7_T2O_General_Purpose_Float_Registers_1_InputAddress_0 AT %IL0: LWORD;
        URIODev1_1_7_T2O_General_Purpose_Float_Registers_1_InputAddress_1 AT %IL8: LWORD;
        URIODev1_1_7_T2O_General_Purpose_Float_Registers_1_InputAddress_2 AT %IL16: LWORD;
        URIODev1_1_7_T2O_General_Purpose_Float_Registers_1_InputAddress_3 AT %IL24: LWORD;
        URIODev1_1_7_T2O_General_Purpose_Float_Registers_1_InputAddress_4 AT %IL32: LWORD;
        URIODev1_1_7_T2O_General_Purpose_Float_Registers_1_InputAddress_5 AT %IL40: LWORD;
        URIODev1_1_7_T2O_General_Purpose_Float_Registers_1_InputAddress_6 AT %IL48: LWORD;
        URIODev1_1_7_T2O_General_Purpose_Float_Registers_1_InputAddress_7 AT %IL56: LWORD;
        URIODev1_1_7_T2O_General_Purpose_Float_Registers_1_InputAddress_8 AT %IL64: LWORD;
        URIODev1_1_7_T2O_General_Purpose_Float_Registers_1_InputAddress_9 AT %IL72: LWORD;
        URIODev1_1_7_T2O_General_Purpose_Float_Registers_1_InputAddress_10 AT %IL80: LWORD;
        URIODev1_1_7_T2O_General_Purpose_Float_Registers_1_InputAddress_11 AT %IL88: LWORD;
        URIODev1_1_8_O2T_Robot_IO_1_OutputAddress_0 AT %QL200: LWORD;
        URIODev1_1_8_O2T_Robot_IO_1_OutputAddress_1 AT %QL208: LWORD;
        URIODev1_1_8_O2T_Robot_IO_1_OutputAddress_2 AT %QL216: LWORD;
        URIODev1_1_9_O2T_General_Purpose_Registers_1_1_OutputAddress_0 AT %QD100: DWORD;
        URIODev1_1_9_O2T_General_Purpose_Registers_1_1_OutputAddress_1 AT %QD104: DWORD;
        URIODev1_1_9_O2T_General_Purpose_Registers_1_1_OutputAddress_2 AT %QD108: DWORD;
        URIODev1_1_9_O2T_General_Purpose_Registers_1_1_OutputAddress_3 AT %QD112: DWORD;
        URIODev1_1_9_O2T_General_Purpose_Registers_1_1_OutputAddress_4 AT %QD116: DWORD;
        URIODev1_1_9_O2T_General_Purpose_Registers_1_1_OutputAddress_5 AT %QD120: DWORD;
        URIODev1_1_9_O2T_General_Purpose_Registers_1_1_OutputAddress_6 AT %QD124: DWORD;
        URIODev1_1_9_O2T_General_Purpose_Registers_1_1_OutputAddress_7 AT %QD128: DWORD;
        URIODev1_1_9_O2T_General_Purpose_Registers_1_1_OutputAddress_8 AT %QD132: DWORD;
        URIODev1_1_9_O2T_General_Purpose_Registers_1_1_OutputAddress_9 AT %QD136: DWORD;
        URIODev1_1_9_O2T_General_Purpose_Registers_1_1_OutputAddress_10 AT %QD140: DWORD;
        URIODev1_1_9_O2T_General_Purpose_Registers_1_1_OutputAddress_11 AT %QD144: DWORD;
        URIODev1_1_9_O2T_General_Purpose_Registers_1_1_OutputAddress_12 AT %QD148: DWORD;
        URIODev1_1_9_O2T_General_Purpose_Registers_1_1_OutputAddress_13 AT %QD152: DWORD;
        URIODev1_1_9_O2T_General_Purpose_Registers_1_1_OutputAddress_14 AT %QD156: DWORD;
        URIODev1_1_9_O2T_General_Purpose_Registers_1_1_OutputAddress_15 AT %QD160: DWORD;
        URIODev1_1_9_O2T_General_Purpose_Registers_1_1_OutputAddress_16 AT %QD164: DWORD;
        URIODev1_1_9_O2T_General_Purpose_Registers_1_1_OutputAddress_17 AT %QD168: DWORD;
        URIODev1_1_9_O2T_General_Purpose_Registers_1_1_OutputAddress_18 AT %QD172: DWORD;
        URIODev1_1_9_O2T_General_Purpose_Registers_1_1_OutputAddress_19 AT %QD176: DWORD;
        URIODev1_1_9_O2T_General_Purpose_Registers_1_1_OutputAddress_20 AT %QD180: DWORD;
        URIODev1_1_9_O2T_General_Purpose_Registers_1_1_OutputAddress_21 AT %QD184: DWORD;
        URIODev1_1_9_O2T_General_Purpose_Registers_1_1_OutputAddress_22 AT %QD188: DWORD;
        URIODev1_1_9_O2T_General_Purpose_Registers_1_1_OutputAddress_23 AT %QD192: DWORD;
        URIODev1_1_9_O2T_General_Purpose_Registers_1_1_OutputAddress_24 AT %QD196: DWORD;
        aventics_Valve_driver_2_valves_1_OutputAddress AT %QB951: BYTE;
        aventics_Valve_driver_3_valves_1_OutputAddress AT %QB954: BYTE;
        aventics_Valve_driver_4_valves_1_OutputAddress AT %QB955: BYTE;
        aventics_Valve_driver_4_valves_2_OutputAddress AT %QB953: BYTE;
        aventics_Valve_driver_4_valves_3_OutputAddress AT %QB952: BYTE;
        cmmtas_DoServo_Submodule_1_InputAddress_0 AT %IL1644: LWORD;
        cmmtas_DoServo_Submodule_1_InputAddress_1 AT %IL1652: LWORD;
        cmmtas_DoServo_Submodule_1_InputAddress_2 AT %IL1660: LWORD;
        cmmtas_DoServo_Submodule_2_InputAddress AT %IW1668: WORD;
        cmmtas_DoServo_Submodule_1_OutputAddress_0 AT %QL1091: LWORD;
        cmmtas_DoServo_Submodule_1_OutputAddress_1 AT %QL1099: LWORD;
        cmmtas_DoServo_Submodule_1_OutputAddress_2 AT %QL1107: LWORD;
        cmmtas_DoServo_Submodule_2_OutputAddress AT %QL1115: LWORD;
        et200sp_CM_4xIO_Link_V2_2_144I_128O_1_InputAddress_0 AT %IL1496: LWORD;
        et200sp_CM_4xIO_Link_V2_2_144I_128O_1_InputAddress_1 AT %IL1504: LWORD;
        et200sp_CM_4xIO_Link_V2_2_144I_128O_1_InputAddress_2 AT %IL1512: LWORD;
        et200sp_CM_4xIO_Link_V2_2_144I_128O_1_InputAddress_3 AT %IL1520: LWORD;
        et200sp_CM_4xIO_Link_V2_2_144I_128O_1_InputAddress_4 AT %IL1528: LWORD;
        et200sp_CM_4xIO_Link_V2_2_144I_128O_1_InputAddress_5 AT %IL1536: LWORD;
        et200sp_CM_4xIO_Link_V2_2_144I_128O_1_InputAddress_6 AT %IL1544: LWORD;
        et200sp_CM_4xIO_Link_V2_2_144I_128O_1_InputAddress_7 AT %IL1552: LWORD;
        et200sp_CM_4xIO_Link_V2_2_144I_128O_1_InputAddress_8 AT %IL1560: LWORD;
        et200sp_CM_4xIO_Link_V2_2_144I_128O_1_InputAddress_9 AT %IL1568: LWORD;
        et200sp_CM_4xIO_Link_V2_2_144I_128O_1_InputAddress_10 AT %IL1576: LWORD;
        et200sp_CM_4xIO_Link_V2_2_144I_128O_1_InputAddress_11 AT %IL1584: LWORD;
        et200sp_CM_4xIO_Link_V2_2_144I_128O_1_InputAddress_12 AT %IL1592: LWORD;
        et200sp_CM_4xIO_Link_V2_2_144I_128O_1_InputAddress_13 AT %IL1600: LWORD;
        et200sp_CM_4xIO_Link_V2_2_144I_128O_1_InputAddress_14 AT %IL1608: LWORD;
        et200sp_CM_4xIO_Link_V2_2_144I_128O_1_InputAddress_15 AT %IL1616: LWORD;
        et200sp_CM_4xIO_Link_V2_2_144I_128O_1_InputAddress_16 AT %IL1624: LWORD;
        et200sp_CM_4xIO_Link_V2_2_144I_128O_1_InputAddress_17 AT %IL1632: LWORD;
        et200sp_CM_4xIO_Link_V2_2_144I_128O_1_OutputAddress_0 AT %QL959: LWORD;
        et200sp_CM_4xIO_Link_V2_2_144I_128O_1_OutputAddress_1 AT %QL967: LWORD;
        et200sp_CM_4xIO_Link_V2_2_144I_128O_1_OutputAddress_2 AT %QL975: LWORD;
        et200sp_CM_4xIO_Link_V2_2_144I_128O_1_OutputAddress_3 AT %QL983: LWORD;
        et200sp_CM_4xIO_Link_V2_2_144I_128O_1_OutputAddress_4 AT %QL991: LWORD;
        et200sp_CM_4xIO_Link_V2_2_144I_128O_1_OutputAddress_5 AT %QL999: LWORD;
        et200sp_CM_4xIO_Link_V2_2_144I_128O_1_OutputAddress_6 AT %QL1007: LWORD;
        et200sp_CM_4xIO_Link_V2_2_144I_128O_1_OutputAddress_7 AT %QL1015: LWORD;
        et200sp_CM_4xIO_Link_V2_2_144I_128O_1_OutputAddress_8 AT %QL1023: LWORD;
        et200sp_CM_4xIO_Link_V2_2_144I_128O_1_OutputAddress_9 AT %QL1031: LWORD;
        et200sp_CM_4xIO_Link_V2_2_144I_128O_1_OutputAddress_10 AT %QL1039: LWORD;
        et200sp_CM_4xIO_Link_V2_2_144I_128O_1_OutputAddress_11 AT %QL1047: LWORD;
        et200sp_CM_4xIO_Link_V2_2_144I_128O_1_OutputAddress_12 AT %QL1055: LWORD;
        et200sp_CM_4xIO_Link_V2_2_144I_128O_1_OutputAddress_13 AT %QL1063: LWORD;
        et200sp_CM_4xIO_Link_V2_2_144I_128O_1_OutputAddress_14 AT %QL1071: LWORD;
        et200sp_CM_4xIO_Link_V2_2_144I_128O_1_OutputAddress_15 AT %QL1079: LWORD;
        et200sp_1_DI_ST_1_InputAddress AT %IB1495: BYTE;
        et200sp_1_DI_ST_2_InputAddress AT %IB1494: BYTE;
        et200sp_1_DQ_ST_1_OutputAddress AT %QB958: BYTE;
        festocpx_MPA1S_VMPA1_FB_EMG_8_1_OutputAddress AT %QB956: BYTE;
        festocpx_MPA1S_VMPA1_FB_EMS_8_OutputAddress AT %QB957: BYTE;
        is7600_Acquisition_Control_OutputAddress AT %QB798: BYTE;
        is7600_Acquisition_Status_InputAddress_0 AT %IB1324: BYTE;
        is7600_Acquisition_Status_InputAddress_1 AT %IB1325: BYTE;
        is7600_Acquisition_Status_InputAddress_2 AT %IB1326: BYTE;
        is7600_Command_Control_InputAddress AT %IW1327: WORD;
        is7600_Command_Control_OutputAddress AT %QW794: WORD;
        is7600_Inspection_Control_OutputAddress AT %QB797: BYTE;
        is7600_Inspection_Status_InputAddress AT %ID1320: DWORD;
        is7600_Result_Data_64_bytes_InputAddress_0 AT %ID1252: DWORD;
        is7600_Result_Data_64_bytes_InputAddress_1 AT %ID1256: DWORD;
        is7600_Result_Data_64_bytes_InputAddress_2 AT %ID1260: DWORD;
        is7600_Result_Data_64_bytes_InputAddress_3 AT %ID1264: DWORD;
        is7600_Result_Data_64_bytes_InputAddress_4 AT %ID1268: DWORD;
        is7600_Result_Data_64_bytes_InputAddress_5 AT %ID1272: DWORD;
        is7600_Result_Data_64_bytes_InputAddress_6 AT %ID1276: DWORD;
        is7600_Result_Data_64_bytes_InputAddress_7 AT %ID1280: DWORD;
        is7600_Result_Data_64_bytes_InputAddress_8 AT %ID1284: DWORD;
        is7600_Result_Data_64_bytes_InputAddress_9 AT %ID1288: DWORD;
        is7600_Result_Data_64_bytes_InputAddress_10 AT %ID1292: DWORD;
        is7600_Result_Data_64_bytes_InputAddress_11 AT %ID1296: DWORD;
        is7600_Result_Data_64_bytes_InputAddress_12 AT %ID1300: DWORD;
        is7600_Result_Data_64_bytes_InputAddress_13 AT %ID1304: DWORD;
        is7600_Result_Data_64_bytes_InputAddress_14 AT %ID1308: DWORD;
        is7600_Result_Data_64_bytes_InputAddress_15 AT %ID1312: DWORD;
        is7600_Result_Data_64_bytes_InputAddress_16 AT %ID1316: DWORD;
        is7600_SoftEvent_Control_InputAddress AT %IB1329: BYTE;
        is7600_SoftEvent_Control_OutputAddress AT %QB796: BYTE;
        is7600_User_Data_64_bytes_OutputAddress_0 AT %QL730: LWORD;
        is7600_User_Data_64_bytes_OutputAddress_1 AT %QL738: LWORD;
        is7600_User_Data_64_bytes_OutputAddress_2 AT %QL746: LWORD;
        is7600_User_Data_64_bytes_OutputAddress_3 AT %QL754: LWORD;
        is7600_User_Data_64_bytes_OutputAddress_4 AT %QL762: LWORD;
        is7600_User_Data_64_bytes_OutputAddress_5 AT %QL770: LWORD;
        is7600_User_Data_64_bytes_OutputAddress_6 AT %QL778: LWORD;
        is7600_User_Data_64_bytes_OutputAddress_7 AT %QL786: LWORD;
        reader_st1_Acquisition_Control_OutputAddress AT %QB940: BYTE;
        reader_st1_Acquisition_Status_InputAddress_0 AT %IB1481: BYTE;
        reader_st1_Acquisition_Status_InputAddress_1 AT %IB1482: BYTE;
        reader_st1_Acquisition_Status_InputAddress_2 AT %IB1483: BYTE;
        reader_st1_Results_Control_OutputAddress AT %QB939: BYTE;
        reader_st1_Results_Status_InputAddress AT %IB1480: BYTE;
        reader_st1_Soft_Event_Control_InputAddress AT %IB1479: BYTE;
        reader_st1_Soft_Event_Control_OutputAddress AT %QB938: BYTE;
        reader_st2_Acquisition_Control_OutputAddress AT %QB869: BYTE;
        reader_st2_Acquisition_Status_InputAddress_0 AT %IB1404: BYTE;
        reader_st2_Acquisition_Status_InputAddress_1 AT %IB1405: BYTE;
        reader_st2_Acquisition_Status_InputAddress_2 AT %IB1406: BYTE;
        reader_st2_Result_Data_64_bytes_InputAddress_0 AT %IL1330: LWORD;
        reader_st2_Result_Data_64_bytes_InputAddress_1 AT %IL1338: LWORD;
        reader_st2_Result_Data_64_bytes_InputAddress_2 AT %IL1346: LWORD;
        reader_st2_Result_Data_64_bytes_InputAddress_3 AT %IL1354: LWORD;
        reader_st2_Result_Data_64_bytes_InputAddress_4 AT %IL1362: LWORD;
        reader_st2_Result_Data_64_bytes_InputAddress_5 AT %IL1370: LWORD;
        reader_st2_Result_Data_64_bytes_InputAddress_6 AT %IL1378: LWORD;
        reader_st2_Result_Data_64_bytes_InputAddress_7 AT %IL1386: LWORD;
        reader_st2_Result_Data_64_bytes_InputAddress_8 AT %IL1394: LWORD;
        reader_st2_Results_Control_OutputAddress AT %QB868: BYTE;
        reader_st2_Results_Status_InputAddress AT %IB1403: BYTE;
        reader_st2_Soft_Event_Control_InputAddress AT %IB1402: BYTE;
        reader_st2_Soft_Event_Control_OutputAddress AT %QB867: BYTE;
        reader_st2_User_Data_64_bytes_OutputAddress_0 AT %QD799: DWORD;
        reader_st2_User_Data_64_bytes_OutputAddress_1 AT %QD803: DWORD;
        reader_st2_User_Data_64_bytes_OutputAddress_2 AT %QD807: DWORD;
        reader_st2_User_Data_64_bytes_OutputAddress_3 AT %QD811: DWORD;
        reader_st2_User_Data_64_bytes_OutputAddress_4 AT %QD815: DWORD;
        reader_st2_User_Data_64_bytes_OutputAddress_5 AT %QD819: DWORD;
        reader_st2_User_Data_64_bytes_OutputAddress_6 AT %QD823: DWORD;
        reader_st2_User_Data_64_bytes_OutputAddress_7 AT %QD827: DWORD;
        reader_st2_User_Data_64_bytes_OutputAddress_8 AT %QD831: DWORD;
        reader_st2_User_Data_64_bytes_OutputAddress_9 AT %QD835: DWORD;
        reader_st2_User_Data_64_bytes_OutputAddress_10 AT %QD839: DWORD;
        reader_st2_User_Data_64_bytes_OutputAddress_11 AT %QD843: DWORD;
        reader_st2_User_Data_64_bytes_OutputAddress_12 AT %QD847: DWORD;
        reader_st2_User_Data_64_bytes_OutputAddress_13 AT %QD851: DWORD;
        reader_st2_User_Data_64_bytes_OutputAddress_14 AT %QD855: DWORD;
        reader_st2_User_Data_64_bytes_OutputAddress_15 AT %QD859: DWORD;
        reader_st2_User_Data_64_bytes_OutputAddress_16 AT %QD863: DWORD;
        rf186c_CM_1_InputAddress AT %IW1642: WORD;
        rf186c_CM_1_OutputAddress AT %QW1089: WORD;
        rf186c_Reader_1_InputAddress AT %IW1640: WORD;
        rf186c_Reader_1_OutputAddress AT %QW1087: WORD;
        wp462_t1_rh_deso_Input_1_byte_1_InputAddress AT %IB1123: BYTE;
        wp462_t1_rh_deso_Input_1_byte_2_InputAddress AT %IB1122: BYTE;
        wp462_t1_rh_deso_Input_1_word_1_InputAddress AT %IW1116: WORD;
        wp462_t1_rh_deso_Input_1_word_2_InputAddress AT %IW1110: WORD;
        wp462_t1_rh_deso_Input_2_word_1_InputAddress AT %ID1118: DWORD;
        wp462_t1_rh_deso_Input_2_word_2_InputAddress AT %ID1112: DWORD;
        wp462_t1_rh_deso_Output_1_byte_1_OutputAddress AT %QB601: BYTE;
        wp462_t1_rh_deso_Output_1_byte_2_OutputAddress AT %QB600: BYTE;

    END_VAR
END_CONFIGURATION
